// TwinCAT 3 PLC project Untitled1
// ProgramVersion: 3.1.4022.0
// libraries:
//   Tc2_Standard, * (Beckhoff Automation GmbH)
//   Tc2_System, * (Beckhoff Automation GmbH)
//   Tc3_Module, * (Beckhoff Automation GmbH)
// project tree:
//   GVLs/ GVLLighting.TcGVL
//   / PlcTask.TcTTO
//   POUs/ MAIN.TcPOU, POURunLight.TcPOU
// real-time tasks:
//   TASK PlcTask: cycle T#1ms, priority 20, ADS port 350

CONFIGURATION Untitled1
    RESOURCE PLC ON TwinCAT3
        TASK PlcTask(INTERVAL := T#1ms, PRIORITY := 20);
        PROGRAM MAIN WITH PlcTask : MAIN;
    END_RESOURCE
END_CONFIGURATION

// ---- GVLs/GVLLighting.TcGVL
{attribute 'qualified_only'}
VAR_GLOBAL
	LightingStatus AT %Q*:BOOL ;
	StartLight AT %I*:BOOL ;
	StopLight AT %I*:BOOL ;
END_VAR

// ---- POUs/MAIN.TcPOU
PROGRAM MAIN
VAR
END_VAR

POURunLight();

END_PROGRAM

// ---- POUs/POURunLight.TcPOU
PROGRAM POURunLight
VAR
END_VAR

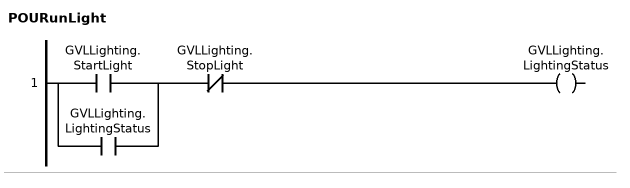
// NETWORK 1
GVLLighting.LightingStatus := (GVLLighting.StartLight OR GVLLighting.LightingStatus) AND NOT GVLLighting.StopLight;

END_PROGRAM
